{attribute addProperty BoxType "EL4712--0000"}
{attribute addProperty Id "Ch1_CycleCountAT %Q*UINT162"}
{attribute addProperty CRC "3106366676"}
{attribute addProperty SizeInBites "16"}
{attribute addProperty SizeInBytes "2"}
TYPE Ch1_CycleCount_B92764D4 :
STRUCT
	{attribute addProperty Name "Ch1_CycleCount"}
	Ch1_CycleCount AT %Q* : UINT;
END_STRUCT
END_TYPE

(* stored: Version 1.2.0.0, ProductVersion 3.1.4024.9
   DUT Ch1_CycleCount_B92764D4: Id {61ee999a-ed9d-4192-ac4c-df0fc7b3124c} *)
